FUNCTION_BLOCK FB_DriveNc EXTENDS FB_DriveBase
VAR_INPUT
END_VAR
VAR_OUTPUT
END_VAR
VAR
END_VAR

METHOD Disable : BOOL
END_METHOD

METHOD Enable : BOOL
END_METHOD

METHOD MoveToPosition : BOOL
END_METHOD

METHOD Reset : BOOL
END_METHOD

END_FUNCTION_BLOCK

(* stored: Version 1.1.0.1, ProductVersion 3.1.4024.6
   POU FB_DriveNc: Id {201d3134-d070-4ef8-af2a-b7d6dbe47945}, SpecialFunc None
   Method Disable: Id {13851cc4-56c5-4b29-8727-b1d38cd557f0}
   Method Enable: Id {363753d5-05d7-4e8c-91d4-2aff5478ccc7}
   Method MoveToPosition: Id {39475d72-7456-4848-911d-0ddb2f34fe01}
   Method Reset: Id {b483f353-b49b-44ef-aecf-993a066705c7} *)
